# EPICS substitutions: evrSupport/Db/evr/evrEventFACET.substitutions
#==============================================================================
#
# Abs:  EVR Event Records
#
# Name: evrEventAll.substitutions
#
#==============================================================================
#
file evrPatternProc.db {
pattern { DEV       }
	{ $(DEVICE) }
}
